Staubli VAL3: HIT_YD.pjx

--- HIT_YD.pjx ---
Parameters version=s7.6.2 stackSize=5000 millimeterUnit=true
Program file=OMAC_Abort.pgx
Program file=OMAC_Hold.pgx
Program file=OMAC_Main.pgx
Program file=OMAC_Reset.pgx
Program file=OMAC_Start.pgx
Program file=OMAC_Stop.pgx
Program file=OMAC_Unhold.pgx
Program file=ServerGet.pgx
Program file=ServerSend.pgx
Program file=blow.pgx
Program file=bypassPick.pgx
Program file=cellManager.pgx
Program file=getToolStatus.pgx
Program file=goHome.pgx
Program file=init.pgx
Program file=initTracking.pgx
Program file=isInSafetyArea.pgx
Program file=ModbusGet.pgx
Program file=modbusSet.pgx
Program file=overflowPick.pgx
Program file=Place.pgx
Program file=productionCycle.pgx
Program file=robot2PC.pgx
Program file=robot2PLC.pgx
Program file=send2NextRob.pgx
Program file=setAlarm.pgx
Program file=setConvSpeed.pgx
Program file=start.pgx
Program file=stop.pgx
Program file=trackErr_init.pgx
Program file=trackingPick.pgx
Program file=transferQueue.pgx
Data file=HIT_YD.dtx
Library alias=mot path=Disk://Tracking/Motion/Motion.pjx autoload=true password=
Type name=object path=Disk://Tracking/Templates/object/object.pjx

--- HIT_YD.dtx ---
aio aConvSpeed = {link=ModbusSrv-0\Modbus-Word\ao[3]}
aio aPlcCmd = {link=ModbusSrv-0\Modbus-Word\ai[0]}
aio aRbAlarm = {link=ModbusSrv-0\Modbus-Word\ao[0]}
aio aRbStatus = {link=ModbusSrv-0\Modbus-Word\ao[1]}
bool _bConvExist = true
bool _bEndCycle
bool _bIsPicking
bool _bIsPlacing
bool _bMutexCnvQueue
bool _bOverflowed = true
bool _bPartInTool = true
bool _bSentToHome
bool _bVisionOK = true
bool bIsConnectPC
bool bLockPage
bool bPickDetection
bool bSetConvSpeed
bool bSyn
bool bTransferData = true
dio dAlarm[8]
  [0] = {link=ModbusSrv-0\Modbus-Bit\do[8]}
  [1] = {link=ModbusSrv-0\Modbus-Bit\do[9]}
  [2] = {link=ModbusSrv-0\Modbus-Bit\do[10]}
  [3] = {link=ModbusSrv-0\Modbus-Bit\do[11]}
  [4] = {link=ModbusSrv-0\Modbus-Bit\do[12]}
  [5] = {link=ModbusSrv-0\Modbus-Bit\do[13]}
  [6] = {link=ModbusSrv-0\Modbus-Bit\do[14]}
  [7] = {link=ModbusSrv-0\Modbus-Bit\do[15]}
dio dBlow = {link=BasicIO-1\%Q5}
dio dConvControl[2]
  [0] = {link=BasicIO-1\%I4}
  [1] = {link=BasicIO-1\%Q6}
dio dPartInTool = {link=fIn0}
dio dPermitPlace[4]
  [0] = {link=BasicIO-1\%I3}
  [1] = {link=BasicIO-1\%I2}
  [2] = {link=BasicIO-1\%I1}
  [3] = {link=BasicIO-1\%I0}
dio dPlaceDone[4]
  [0] = {link=BasicIO-1\%Q11}
  [1] = {link=BasicIO-1\%Q10}
  [2] = {link=BasicIO-1\%Q9}
  [3] = {link=BasicIO-1\%Q8}
dio dStartControl[4]
  [0] = {link=ModbusSrv-0\Modbus-Bit\di[4]}
  [1] = {link=ModbusSrv-0\Modbus-Bit\di[5]}
  [2] = {link=ModbusSrv-0\Modbus-Bit\di[6]}
  [3] = {link=ModbusSrv-0\Modbus-Bit\di[7]}
dio dStartState[4]
  [0] = {link=ModbusSrv-0\Modbus-Bit\do[4]}
  [1] = {link=ModbusSrv-0\Modbus-Bit\do[5]}
  [2] = {link=ModbusSrv-0\Modbus-Bit\do[6]}
  [3] = {link=ModbusSrv-0\Modbus-Bit\do[7]}
dio dVacuum = {link=BasicIO-1\%Q4}
frame fConveyor = {x=365.904087, y=326.91934, z=-82.602337, rx=-0.010861, ry=-0.059106, rz=0.004608, fatherId=world[0]}
frame fDetection = {x=392.598601, y=461.346273, z=-82.976862, rx=0.205045, ry=0.617271, rz=0.011036, fatherId=world[0]}
jointRs jDropPart = {j1=102.785955, j2=-95.43121, j3=69.578977, j4=134.260732}
jointRs jHome = {j1=102.785955, j2=-95.43121, j3=69.578977, j4=134.260732}
jointRs jPark = {j1=102.785955, j2=-95.43121, j3=69.578977, j4=134.260732}
mdesc _mLoad = {accel=133.4025, vel=115.5, decel=133.4025}
mdesc mLoad = {accel=121, vel=110, decel=121}
mdesc mNomSpeed = {accel=144, vel=120, decel=144, leave=20, reach=20}
mdesc mPickDown = {accel=144, vel=120, decel=144, blend=off, leave=10, reach=10}
mdesc mPickup = {accel=121, vel=110, decel=121, leave=40, reach=40}
mdesc mPlaceDown = {accel=144, vel=120, decel=144, blend=off, leave=15, reach=15}
mdesc mPlaceUp = {accel=144, vel=120, decel=144, blend=cartesian, leave=20, reach=20}
mdesc mSlow = {accel=1, vel=10, decel=1, leave=10, reach=10}
mdesc mUnload = {accel=144, vel=120, decel=144, leave=40, reach=40}
num _nBlowDelay
num _nCntBypassed = 1
num _nCntPartsDone[2]
  [0] = 74956
  [1] = 74907
num _nCntTransfered = 8
num _nConvSpd
num _nCycleTime[4]
  [0] = 33.16
  [1] = 2.331
  [2] = 48.87
  [3] = 0.935
num _nCycleTimeIndx
num _nID = -1
num _nLastStateCMD
num _nOmacStat = 3
num _nPartID = 1
num _nPlaceCurItem[2]
num _nPullIndexTQ = 8
num _nPushIndexTQ = 8
num _nStateCMD
num _nTimer = 355.546
num _nTrackErr = 315
num nBlowID = 0.3
num nBypass = 1
num nLoadRatio[4]
  [0] = 0.7
  [1] = 0.85
  [2] = 0.95
  [3] = 1.05
num nNomConvSpeed = 100
num nPartHeight = 6
num nPickAppro = 65
num nPickOS_X = -3
num nPickOS_Y
num nPlaceAppro = 60
public num nPlaceNum = 3
num nSafeMaxX = 850
num nSafeMaxY = 650
num nSafeMinX
num nSafeMinY
num nStopTime = 0.02
num nTestData[5]
  [0] = 6
  [1] = -49
  [2] = 55
  [4] = 24206
num nVacuumID
num nWaitDist2Up4BP = -300
num nWaitDistToDown = 50
num nWaitDistToUp[1 3]
  [0,0] = -80
  [0,1] = 120
  [0,2] = 400
num nWaitDistX
object _oTransferQueue[1 100]
  [0,0]
    num nID = -1
    num nLatchedValue
    trsf trTrsf
  [0,1]
    num nID = -1
    num nLatchedValue
    trsf trTrsf
  [0,2]
    num nID = -1
    num nLatchedValue
    trsf trTrsf
  [0,3]
    num nID = -1
    num nLatchedValue
    trsf trTrsf
  [0,4]
    num nID = -1
    num nLatchedValue
    trsf trTrsf
  [0,5]
    num nID = -1
    num nLatchedValue
    trsf trTrsf
  [0,6]
    num nID = -1
    num nLatchedValue
    trsf trTrsf
  [0,7]
    num nID = -1
    num nLatchedValue
    trsf trTrsf
  [0,8]
    num nID = -1
    num nLatchedValue
    trsf trTrsf
  [0,9]
    num nID = -1
    num nLatchedValue
    trsf trTrsf
  [0,10]
    num nID = -1
    num nLatchedValue
    trsf trTrsf
  [0,11]
    num nID = -1
    num nLatchedValue
    trsf trTrsf
  [0,12]
    num nID = -1
    num nLatchedValue
    trsf trTrsf
  [0,13]
    num nID = -1
    num nLatchedValue
    trsf trTrsf
  [0,14]
    num nID = -1
    num nLatchedValue
    trsf trTrsf
  [0,15]
    num nID = -1
    num nLatchedValue
    trsf trTrsf
  [0,16]
    num nID = -1
    num nLatchedValue
    trsf trTrsf
  [0,17]
    num nID = -1
    num nLatchedValue
    trsf trTrsf
  [0,18]
    num nID = -1
    num nLatchedValue
    trsf trTrsf
  [0,19]
    num nID = -1
    num nLatchedValue
    trsf trTrsf
  [0,20]
    num nID = -1
    num nLatchedValue
    trsf trTrsf
  [0,21]
    num nID = -1
    num nLatchedValue
    trsf trTrsf
  [0,22]
    num nID = -1
    num nLatchedValue
    trsf trTrsf
  [0,23]
    num nID = -1
    num nLatchedValue
    trsf trTrsf
  [0,24]
    num nID = -1
    num nLatchedValue
    trsf trTrsf
  [0,25]
    num nID = -1
    num nLatchedValue
    trsf trTrsf
  [0,26]
    num nID = -1
    num nLatchedValue
    trsf trTrsf
  [0,27]
    num nID = -1
    num nLatchedValue
    trsf trTrsf
  [0,28]
    num nID = -1
    num nLatchedValue
    trsf trTrsf
  [0,29]
    num nID = -1
    num nLatchedValue
    trsf trTrsf
  [0,30]
    num nID = -1
    num nLatchedValue
    trsf trTrsf
  [0,31]
    num nID = -1
    num nLatchedValue
    trsf trTrsf
  [0,32]
    num nID = -1
    num nLatchedValue
    trsf trTrsf
  [0,33]
    num nID = -1
    num nLatchedValue
    trsf trTrsf
  [0,34]
    num nID = -1
    num nLatchedValue
    trsf trTrsf
  [0,35]
    num nID = -1
    num nLatchedValue
    trsf trTrsf
  [0,36]
    num nID = -1
    num nLatchedValue
    trsf trTrsf
  [0,37]
    num nID = -1
    num nLatchedValue
    trsf trTrsf
  [0,38]
    num nID = -1
    num nLatchedValue
    trsf trTrsf
  [0,39]
    num nID = -1
    num nLatchedValue
    trsf trTrsf
  [0,40]
    num nID = -1
    num nLatchedValue
    trsf trTrsf
  [0,41]
    num nID = -1
    num nLatchedValue
    trsf trTrsf
  [0,42]
    num nID = -1
    num nLatchedValue
    trsf trTrsf
  [0,43]
    num nID = -1
    num nLatchedValue
    trsf trTrsf
  [0,44]
    num nID = -1
    num nLatchedValue
    trsf trTrsf
  [0,45]
    num nID = -1
    num nLatchedValue
    trsf trTrsf
  [0,46]
    num nID = -1
    num nLatchedValue
    trsf trTrsf
  [0,47]
    num nID = -1
    num nLatchedValue
    trsf trTrsf
  [0,48]
    num nID = -1
    num nLatchedValue
    trsf trTrsf
  [0,49]
    num nID = -1
    num nLatchedValue
    trsf trTrsf
  [0,50]
    num nID = -1
    num nLatchedValue
    trsf trTrsf
  [0,51]
    num nID = -1
    num nLatchedValue
    trsf trTrsf
  [0,52]
    num nID = -1
    num nLatchedValue
    trsf trTrsf
  [0,53]
    num nID = -1
    num nLatchedValue
    trsf trTrsf
  [0,54]
    num nID = -1
    num nLatchedValue
    trsf trTrsf
  [0,55]
    num nID = -1
    num nLatchedValue
    trsf trTrsf
  [0,56]
    num nID = -1
    num nLatchedValue
    trsf trTrsf
  [0,57]
    num nID = -1
    num nLatchedValue
    trsf trTrsf
  [0,58]
    num nID = -1
    num nLatchedValue
    trsf trTrsf
  [0,59]
    num nID = -1
    num nLatchedValue
    trsf trTrsf
  [0,60]
    num nID = -1
    num nLatchedValue
    trsf trTrsf
  [0,61]
    num nID = -1
    num nLatchedValue
    trsf trTrsf
  [0,62]
    num nID = -1
    num nLatchedValue
    trsf trTrsf
  [0,63]
    num nID = -1
    num nLatchedValue
    trsf trTrsf
  [0,64]
    num nID = -1
    num nLatchedValue
    trsf trTrsf
  [0,65]
    num nID = -1
    num nLatchedValue
    trsf trTrsf
  [0,66]
    num nID = -1
    num nLatchedValue
    trsf trTrsf
  [0,67]
    num nID = -1
    num nLatchedValue
    trsf trTrsf
  [0,68]
    num nID = -1
    num nLatchedValue
    trsf trTrsf
  [0,69]
    num nID = -1
    num nLatchedValue
    trsf trTrsf
  [0,70]
    num nID = -1
    num nLatchedValue
    trsf trTrsf
  [0,71]
    num nID = -1
    num nLatchedValue
    trsf trTrsf
  [0,72]
    num nID = -1
    num nLatchedValue
    trsf trTrsf
  [0,73]
    num nID = -1
    num nLatchedValue
    trsf trTrsf
  [0,74]
    num nID = -1
    num nLatchedValue
    trsf trTrsf
  [0,75]
    num nID = -1
    num nLatchedValue
    trsf trTrsf
  [0,76]
    num nID = -1
    num nLatchedValue
    trsf trTrsf
  [0,77]
    num nID = -1
    num nLatchedValue
    trsf trTrsf
  [0,78]
    num nID = -1
    num nLatchedValue
    trsf trTrsf
  [0,79]
    num nID = -1
    num nLatchedValue
    trsf trTrsf
  [0,80]
    num nID = -1
    num nLatchedValue
    trsf trTrsf
  [0,81]
    num nID = -1
    num nLatchedValue
    trsf trTrsf
  [0,82]
    num nID = -1
    num nLatchedValue
    trsf trTrsf
  [0,83]
    num nID = -1
    num nLatchedValue
    trsf trTrsf
  [0,84]
    num nID = -1
    num nLatchedValue
    trsf trTrsf
  [0,85]
    num nID = -1
    num nLatchedValue
    trsf trTrsf
  [0,86]
    num nID = -1
    num nLatchedValue
    trsf trTrsf
  [0,87]
    num nID = -1
    num nLatchedValue
    trsf trTrsf
  [0,88]
    num nID = -1
    num nLatchedValue
    trsf trTrsf
  [0,89]
    num nID = -1
    num nLatchedValue
    trsf trTrsf
  [0,90]
    num nID = -1
    num nLatchedValue
    trsf trTrsf
  [0,91]
    num nID = -1
    num nLatchedValue
    trsf trTrsf
  [0,92]
    num nID = -1
    num nLatchedValue
    trsf trTrsf
  [0,93]
    num nID = -1
    num nLatchedValue
    trsf trTrsf
  [0,94]
    num nID = -1
    num nLatchedValue
    trsf trTrsf
  [0,95]
    num nID = -1
    num nLatchedValue
    trsf trTrsf
  [0,96]
    num nID = -1
    num nLatchedValue
    trsf trTrsf
  [0,97]
    num nID = -1
    num nLatchedValue
    trsf trTrsf
  [0,98]
    num nID = -1
    num nLatchedValue
    trsf trTrsf
  [0,99]
    num nID = -1
    num nLatchedValue
    trsf trTrsf
pointRs pPick = {shoulder=lefty, fatherId=fDetection[0]}
pointRs pPlace[4]
  [0] = {x=356.46, y=115, z=-70.81, rx=180, rz=-98.019983, shoulder=lefty, fatherId=world[0]}
  [1] = {x=486.131736, y=115, z=-70.81, rx=180, rz=-98.021161, shoulder=lefty, fatherId=world[0]}
  [2] = {x=630, y=105, z=-70.81, rx=180, rz=-98.02183, shoulder=lefty, fatherId=world[0]}
  [3] = {x=770, y=105, z=-70.8, rx=180, rz=-98.02084, shoulder=lefty, fatherId=world[0]}
sio skToRobot = {link=Socket\toRobot_sk1}
sio sktoPC = {link=Socket\toPC}
sio synServer = {link=Socket\synRobot1}
string _sCycleStatus = "Distance to pick:  -79.66"
string sConveyorList = "cvIn"
string sDataPC = "stop"
string sString = "done"
tool tGripper = {z=85, rz=45, fatherId=flange[0], ioLink=valve1}

--- cellManager.pgx ---
program cellManager()
  local joint l_jHere
  local num l_nConvSpeedOld
  local num l_nErr
  local num l_nI
begin
  // This program is the cell manager, it manage:
  //  -  Variable initializing
  //  -  Launch Tracking
  //  -  Arm Power
  //  -  Robot home position
  //  -  Launch user’s tasks, kills and re-launch user’s task in case of tracking error
  //  -  Displays cycle times and counters.
  //
  // Input parameters
  //  None            :
  //
  // Output parameters
  //  None            :
  //
  //----------------------------------------------------------------
  //

  //  //Launch queue transfer tasks
  //  if _bTransferData[0]
  //    taskCreate "TransferQueue1",100,transferQueue(0)
  //  endIf
  //  // Task to remove picking positions that have pass the downstream limit while the robot is placing a part.
  //  taskCreate "overflowPick",100,overflowPick()

  // Task for production cycle
  if taskStatus("productionCycle")>=0
    taskKill("productionCycle")
  endIf
  wait(taskStatus("productionCycle")<0)
  taskCreate "productionCycle",100,productionCycle()

  //
  if taskStatus("robot2PLC")>=0
    taskKill("robot2PLC")
  endIf
  wait(taskStatus("robot2PLC")<0)
  taskCreate "robot2PLC",100,robot2PLC()

  // Task to set the blow on the tool for a defined period of time
  if taskStatus("blow")>=0
    taskKill("blow")
  endIf
  wait(taskStatus("blow")<0)
  taskCreate "blow",100,blow()
  wait(taskStatus("blow")==1)
  //
  //OMAC进程:Running
  _nOmacStat=3

  //
  //  //Init conveyor speed
  //  call setConvSpeed(0,nNomConvSpeed[0])
  //  l_nConvSpeedOld[0]=nNomConvSpeed[0]
  //
  // Main loop
  do
    if taskStatus("productionCycle")!=1
      taskKill("productionCycle")
      _bMutexCnvQueue=false
      wait(taskStatus("productionCycle")<0)
      taskCreate "productionCycle",100,productionCycle()
    endIf
    // Enable Power
    if isPowered()==false and esStatus()!=2
      if _nOmacStat==3
        enablePower()
        delay(0.5)
      endIf
    endIf
    //
    // Set conveyor speed to the nominal value if the conveyor speed is not controlled by the tasks
    //  overflowPick and overflowPlace
    if bSetConvSpeed[0]
      l_nConvSpeedOld[0]=0
    else
      if l_nConvSpeedOld[0]!=nNomConvSpeed[0]
        call setConvSpeed(0,nNomConvSpeed[0])
        l_nConvSpeedOld[0]=nNomConvSpeed[0]
      endIf
    endIf

    if _nOmacStat==3
      //task TransferQueue1 error management,auto recover
      if bTransferData[0]
        if taskStatus("TransferQueue1")!=1
          logMsg("TransferQueue1任务错误")
          taskKill("TransferQueue1")
          wait(taskStatus("TransferQueue1")==-1)
          taskCreate "TransferQueue1",100,transferQueue(0)
          wait(taskStatus("TransferQueue1")==1)
          logMsg("TransferQueue1自动恢复")
        endIf
      endIf
      //task TransferQueue1 error management,auto recover
      if taskStatus("overflowPick")!=1
        logMsg("overflowPick任务错误")
        taskKill("overflowPick")
        wait(taskStatus("overflowPick")==-1)
        taskCreate "overflowPick",100,overflowPick()
        wait(taskStatus("overflowPick")==1)
        logMsg("overflowPick自动恢复")
      endIf
      // Tracking error management
      if isSettled()==true and $trackingState()==-1
        if _nOmacStat==3
          if _bIsPicking==true
            logMsg("抓取时跟踪错误")
          endIf
          if _bIsPlacing==true
            logMsg("放件时运动错误")
          endIf
          //记录跟踪错误次数
          _nTrackErr=_nTrackErr+1
          stopMove()
          resetMotion()
          call trackErr_init()
          autoConnectMove(true)
          l_jHere=herej()
          l_jHere.j3=jHome.j3
          movej(l_jHere,tGripper,mNomSpeed)
          movej(jHome,tGripper,mNomSpeed)
          _bSentToHome=true
          //          //Launch queue transfer tasks
          //          if _bTransferData[0]
          //            taskCreate "TransferQueue1",100,transferQueue(0)
          //          endIf
          //          // Task to remove picking positions that have pass the downstream limit while the robot is placing a part.
          //          taskCreate "overflowPick",100,overflowPick()
          // Task for production cycle

          if taskStatus("productionCycle")>=0
            taskKill("productionCycle")
          endIf
          wait(taskStatus("productionCycle")<0)
          taskCreate "productionCycle",100,productionCycle()
          wait(taskStatus("productionCycle")==1)
        endIf
      endIf
    endIf
    //show cv speed
    if _bConvExist
      call mot:getConvSpeed(0,_nConvSpd,l_nErr)
      gotoxy(0,0)
      put("                    ")
      gotoxy(0,0)
      put("传送带速度："+toString("",_nConvSpd)+" mm/s")
    endIf



    if isSettled()==true and isEmpty()==false
      //restartMove()
    endIf
    delay(0)
  until false
end

--- isInSafetyArea.pgx ---
program isInSafetyArea()
  local jointRs l_jHere
  local num l_ns
  local pointRs l_pCurrent
begin
  bIsConnectPC=false
  do
    l_pCurrent=here(flange,world)
    //**************************************************//
    //******** 用来判断机器人是否在安全工作空间 ********//
    //**************************************************//
    if (l_pCurrent.trsf.y>=nSafeMaxY or l_pCurrent.trsf.y<=nSafeMinY or l_pCurrent.trsf.x>=nSafeMaxX or l_pCurrent.trsf.x<=nSafeMinX) and _nOmacStat==3
      aioSet(aRbAlarm,10)
      call setAlarm(7)
      popUpMsg("机器人超出安全工作空间！")
      logMsg("机器人超出安全工作空间！")
      call OMAC_Abort()
    endIf

    if (dConvControl[0]==true)
      dConvControl[1]=true
    else
      dConvControl[1]=false
    endIf

    if (bIsConnectPC==true)
      if (sDataPC=="stop")
        l_ns=clock()
        do
          call setAlarm(0)
        until (clock()-l_ns>0.5)
        call setAlarm(10)
        sDataPC="alarm0"
        bIsConnectPC=false
      endIf
    endIf
    delay(0)
  until false
end

--- ModbusGet.pgx ---
program modbusGet(num& x_nResult (dimensions=1))
begin
  if (dStartControl[1]==true and dStartControl[2]==false and dStartControl[3]==false)
    x_nResult=1
  elseIf (dStartControl[1]==false and dStartControl[2]==true and dStartControl[3]==false)
    x_nResult=2
  elseIf (dStartControl[1]==false and dStartControl[2]==false and dStartControl[3]==true)
    x_nResult=3
  else
    x_nResult=0
  endIf
end

--- OMAC_Abort.pgx ---
program OMAC_Abort()
begin
  //OMAC进程:aborting
  _nOmacStat=10
  logMsg("上位机手动操作：急停")
  resetMotion()
  stopMove()

  call setAlarm(10)
  // Stop task

  taskKill("cellManager")
  taskKill("overflowPick")
  taskKill("productionCycle")
  taskKill("Reset")
  taskKill("Start")
  taskKill("Hold")
  taskKill("Unhold")
  taskKill("Stop")
  taskKill("TransferQueue1")
  taskKill("robot2PLC")
  taskKill("robot2PC")

  wait(isSettled())
  wait(taskStatus("Reset")==-1)
  wait(taskStatus("Start")==-1)
  wait(taskStatus("Hold")==-1)
  wait(taskStatus("Unhold")==-1)
  wait(taskStatus("Stop")==-1)
  wait(taskStatus("cellManager")==-1)
  wait(taskStatus("TransferQueue1")==-1)
  wait(taskStatus("overflowPick")==-1)
  wait(taskStatus("productionCycle")==-1)

  if _bConvExist
    call mot:kill()
    _bConvExist=false
  endIf
  disablePower()
  wait(isPowered()==false)
  //OMAC进程:Stopped
  _nOmacStat=9
  delay(0)
end

--- OMAC_Reset.pgx ---
program OMAC_Reset()
  local bool l_bResult
  local joint l_jHere
  local num l_nKey
begin

  //OMAC进程:resetting
  _nOmacStat=4
  logMsg("上位机手动操作：复位")



  // Reset conveyor speed
  //  call setConvSpeed(0,0)
  //start vision
  _bVisionOK=false
  if taskStatus("robot2PC")>=0
    taskKill("robot2PC")
  endIf
  wait(taskStatus("robot2PC")<0)
  taskCreate "robot2PC",100,robot2PC()
  //wait vision ok
  l_bResult=watch(_bVisionOK,5)
  if l_bResult==false
    //alarm
    logMsg("vision start failed")
    taskKill("robot2PC")
    _nOmacStat=9
    return
  endIf
  // Variable initializing
  call init()
  call trackErr_init()
  // Launch Tracking
  call initTracking()
  if !isInRange(herej())
    aioSet(aRbAlarm,20)
    call setAlarm(1)
    popUpMsg("机器人关节超限!")
    taskCreate "Abort",100,OMAC_Abort()
    return
  endIf
  //
  resetMotion()
  // Enables arm power
  while !isPowered()
    enablePower()
    delay(1)
  endWhile
  _bSentToHome=true
  // Send robot to home position
  l_jHere=herej()
  l_jHere.j3=jHome.j3
  movej(l_jHere,tGripper,mSlow)
  movej(jHome,tGripper,mSlow)
  //
  //
  // Init user screen
  cls()
  gotoxy(0,4)
  put("Cycle Time (Last):    ")
  gotoxy(0,6)
  put("Cycle Time (Average): ")
  gotoxy(0,8)
  put("Cycle Time (Best):    ")
  gotoxy(0,10)
  put("      Pick                Place         ")
  gotoxy(0,11)
  put("  Done   Transfer      Done   ")


  //Launch queue transfer tasks
  if bTransferData[0]
    if taskStatus("TransferQueue1")>=0
      taskKill("TransferQueue1")
    endIf
    taskCreate "TransferQueue1",100,transferQueue(0)
    wait(taskStatus("TransferQueue1")==1)
  endIf

  // Task to remove picking positions that have pass the downstream limit while the robot is placing a part.
  if taskStatus("overflowPick")>=0
    taskKill("overflowPick")
  endIf
  taskCreate "overflowPick",100,overflowPick()
  wait(taskStatus("overflowPick")==1)

  //OMAC进程:ready
  _nOmacStat=1
  delay(0)
end

--- OMAC_Stop.pgx ---
program OMAC_Stop()
  local joint l_jHere
  local string l_sToolStatus
begin

  //OMAC进程:Stopping
  _nOmacStat=8
  logMsg("上位机手动操作：停止")
  stopMove()
  resetMotion()
  //
  // Stop task

  taskKill("cellManager")
  taskKill("overflowPick")
  taskKill("productionCycle")
  taskKill("Reset")
  taskKill("Start")
  taskKill("Hold")
  taskKill("Unhold")
  taskKill("Preheat")
  taskKill("openPallet")
  taskKill("changeBox")
  taskKill("convStopCheck")
  taskKill("TransferQueue1")
  taskKill("robot2PC")
  taskKill("robot2PLC")


  resetMotion()
  while !isPowered()
    enablePower()
    delay(1)
  endWhile
  //
  // Move up axis 3
  l_jHere=herej()
  l_jHere.j3=95
  movej(l_jHere,tGripper,mSlow)
  //
  // Drop the part on the tool
  if bPickDetection==true
    call getToolStatus(l_sToolStatus)
  endIf
  if l_sToolStatus=="PartInTool" or !bPickDetection
    movej(jDropPart,tGripper,mSlow)
    waitEndMove()
    dVacuum=false
  else
    dVacuum=false
  endIf
  //
  // Go to park position
  movej(jPark,tGripper,mSlow)
  waitEndMove()
  wait(taskStatus("Reset")==-1)
  wait(taskStatus("Start")==-1)
  wait(taskStatus("Hold")==-1)
  wait(taskStatus("Unhold")==-1)
  wait(taskStatus("Preheat")==-1)
  wait(taskStatus("openPallet")==-1)
  wait(taskStatus("changeBox")==-1)
  wait(taskStatus("convStopCheck")==-1)
  wait(taskStatus("cellManager")==-1)
  wait(taskStatus("TransferQueue1")==-1)
  wait(taskStatus("overflowPick")==-1)
  wait(taskStatus("productionCycle")==-1)

  if _bConvExist
    call mot:kill()
    _bConvExist=false
  endIf

  disablePower()
  wait(isPowered()==false)
  //OMAC进程:Stopped
  _nOmacStat=9

  delay(0)
end

--- Place.pgx ---
program place()
  local bool l_bNoError
  local joint l_jAppro
  local num l_nConvNum
  local num l_nError
  local num l_nMoveID
  local num l_nTrackStatus
  local pointRs l_pAppro
  local pointRs l_pPlace
  local string l_sToolStatus
begin
  l_nConvNum=1
  link(l_pPlace,world)
  //che modify start
  if nPlaceNum<0
    nPlaceNum=3
  endIf
  _mLoad=mLoad
  _mLoad.vel=mLoad.vel*nLoadRatio[nPlaceNum]
  _mLoad.accel=mLoad.accel*nLoadRatio[nPlaceNum]*nLoadRatio[nPlaceNum]
  _mLoad.decel=mLoad.decel*nLoadRatio[nPlaceNum]*nLoadRatio[nPlaceNum]

  //dControlVacuum[nPlaceNum]=false
  l_pPlace=pPlace[nPlaceNum]
  //end
  // Place part
  l_pAppro=appro(l_pPlace,{0,0,-nPlaceAppro,0,0,0})
  l_bNoError=pointToJoint(tGripper,jHome,l_pAppro,l_jAppro)
  call mot:getTrackStatus(l_nTrackStatus)
  if l_nTrackStatus>0
    // Use trackOff if the robot is synchronized
    if l_bNoError
      call mot:trackOffJ(l_jAppro,tGripper,_mLoad,l_nMoveID,l_nError)
    else
      call mot:trackOff(l_pAppro,tGripper,_mLoad,l_nMoveID,l_nError)
    endIf
  else
    // Use movej if the robot is not synchronized
    if l_bNoError
      l_nMoveID=movej(l_jAppro,tGripper,_mLoad)
    else
      l_nMoveID=movej(l_pAppro,tGripper,_mLoad)
    endIf
  endIf
  // wait permit signal
  //
  wait(dPermitPlace[nPlaceNum]==true)
  l_nMoveID=movel(l_pPlace,tGripper,mPlaceDown)
  wait(getMoveId()>l_nMoveID+nBlowID)
  _nBlowDelay=0.3
  waitEndMove()
  delay(nStopTime)
  l_nMoveID=movel(l_pAppro,tGripper,mPlaceUp)
  // check PartInTool if bPickDetection
  if bPickDetection
    //wait(getMoveId()>l_nMoveID-0.8)
    wait(getMoveId()>l_nMoveID+nBlowID-1.2)
    call getToolStatus(l_sToolStatus)
  else
    //wait(getMoveId()>l_nMoveID-0.2)
    wait(getMoveId()>l_nMoveID+nBlowID-1.2)
    _bPartInTool=false
  endIf
  // send done signal
  //dPlaceDone[nPlaceNum]=true
  wait(getMoveId()>l_nMoveID+0.1)
  delay(0)
  //dPlaceDone[nPlaceNum]=false
  if l_sToolStatus=="PartInTool" or _bPartInTool==false
    // A part has been placed
    _nCntPartsDone[l_nConvNum]=_nCntPartsDone[l_nConvNum]+1
  endIf
  delay(0)

  dPlaceDone[nPlaceNum]=true
  wait(getMoveId()>l_nMoveID+0.4)
  if nPlaceNum==3 and bSyn
    do
      sString=synServer
    until (sString=="done")
  endIf
  if nPlaceNum==0
    //synServer="done"
  endIf
  nPlaceNum=nPlaceNum-1
  nTestData[4]=nTestData[4]+1
  //end

end

--- setAlarm.pgx ---
program setAlarm(num x_nNum (dimensions=1))
begin
  if (x_nNum==0)
    dAlarm[0]=true
    dAlarm[1]=false
    dAlarm[2]=false
    dAlarm[3]=false
    dAlarm[4]=false
    dAlarm[5]=false
    dAlarm[6]=false
    dAlarm[7]=false
  elseIf (x_nNum==1)
    dAlarm[0]=false
    dAlarm[1]=true
    dAlarm[2]=false
    dAlarm[3]=false
    dAlarm[4]=false
    dAlarm[5]=false
    dAlarm[6]=false
    dAlarm[7]=false
  elseIf (x_nNum==2)
    dAlarm[0]=false
    dAlarm[1]=false
    dAlarm[2]=true
    dAlarm[3]=false
    dAlarm[4]=false
    dAlarm[5]=false
    dAlarm[6]=false
    dAlarm[7]=false
  elseIf (x_nNum==3)
    dAlarm[0]=false
    dAlarm[1]=false
    dAlarm[2]=true
    dAlarm[3]=false
    dAlarm[4]=false
    dAlarm[5]=false
    dAlarm[6]=false
    dAlarm[7]=false
  elseIf (x_nNum==4)
    dAlarm[0]=false
    dAlarm[1]=false
    dAlarm[2]=false
    dAlarm[3]=false
    dAlarm[4]=true
    dAlarm[5]=false
    dAlarm[6]=false
    dAlarm[7]=false
  elseIf (x_nNum==5)
    dAlarm[0]=false
    dAlarm[1]=false
    dAlarm[2]=false
    dAlarm[3]=false
    dAlarm[4]=false
    dAlarm[5]=true
    dAlarm[6]=false
    dAlarm[7]=false
  elseIf (x_nNum==6)
    dAlarm[0]=false
    dAlarm[1]=false
    dAlarm[2]=false
    dAlarm[3]=false
    dAlarm[4]=false
    dAlarm[5]=false
    dAlarm[6]=true
    dAlarm[7]=false
  elseIf (x_nNum==7)
    dAlarm[0]=false
    dAlarm[1]=false
    dAlarm[2]=false
    dAlarm[3]=false
    dAlarm[4]=false
    dAlarm[5]=false
    dAlarm[6]=false
    dAlarm[7]=true
  else

    dAlarm[0]=false
    dAlarm[1]=false
    dAlarm[2]=false
    dAlarm[3]=false
    dAlarm[4]=false
    dAlarm[5]=false
    dAlarm[6]=false
  endIf
end
